RoboDK station: AQIS.rdk

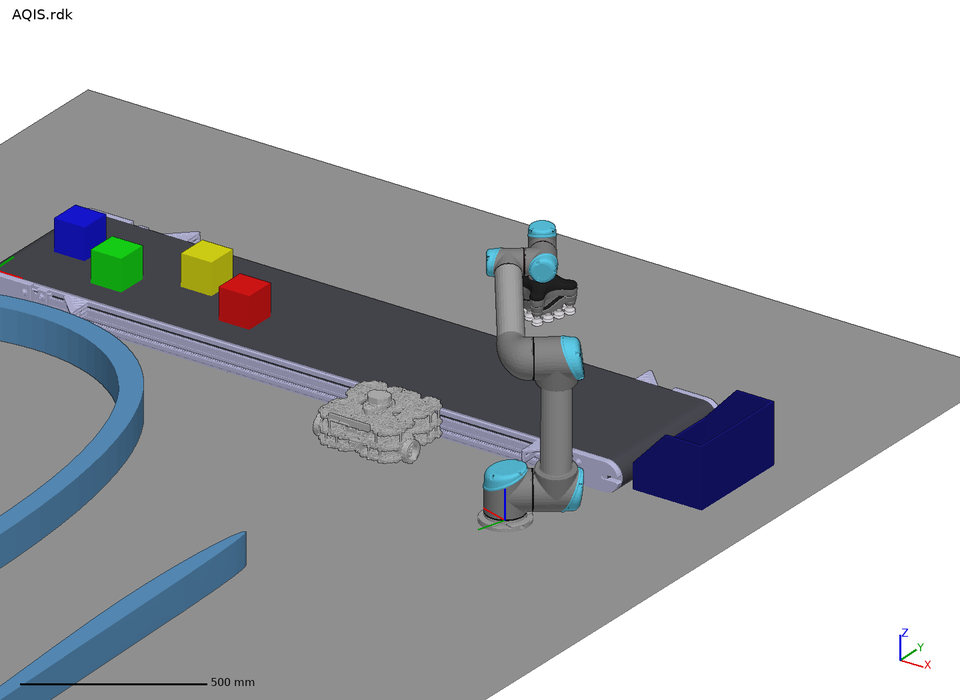
[picture v0: the station drawn from its stored meshes, robots at their saved joint values, targets as dots, program paths as lines]
Station AQIS (saved by RoboDK 5.7.4). Poses are relative to the parent item; angles as X-Y-Z fixed-axis rotations.
  - frame Main at (0, 0, 0) mm
    - frame Conveyor Belt (2m) Base at (0, 1000, 20) mm
      - robot Conveyor Belt (2m): 1 axes
          modified DH rows (alpha deg, a mm, theta deg, d mm): 0, 0, 0, 0 linear
          base shift (0, 0, 0) mm, rotated rx 0 ry 90 rz 0 deg
          joint limits [-500000] to [500000]; home [0]; saved at [0]
    - object Bin Blue at (2060, 1370, -70) mm, rotated rx 0 ry 0 rz -180 deg, size 225 x 337.5 x 191.2 mm, geometry from Bin-Blue.sld
    - object Bin Red at (130, -1910, 0) mm, rotated rx 0 ry 0 rz 90 deg, size 225 x 337.5 x 191.2 mm, geometry from Bin-Red.sld
    - object Blue at (120, 1230, 20) mm, size 100 x 100 x 100 mm, geometry from Blue.step
    - object Green at (310, 1130, 20) mm, size 100 x 100 x 100 mm, geometry from Green.step
    - object Red at (720, 1140, 20) mm, size 100 x 100 x 100 mm, geometry from Red.step
    - object Yellow at (520, 1250, 20) mm, size 100 x 100 x 100 mm, geometry from Yellow.step
    - frame UR5 Base at (1880.84, 695.53, -76.85) mm, rotated rx 0 ry 0 rz 163.4 deg
      - robot UR5: 6 axes
          modified DH rows (alpha deg, a mm, theta deg, d mm): 0, 0, 0, 89.2; 90, 0, 180, 0; 0, 425, 0, 0; 0, 392, 0, 109.3; -90, 0, 0, 94.75; 90, 0, 180, 82.5
          joint limits [-360, -360, -360, -360, -360, -360] to [360, 360, 360, 360, 360, 360]; home [0, -90, -90, 0, 90, 0]; saved at [-36.82, -81.705, -83.159, -101.079, 89.606, 237.429]
        - tool OnRobot VG10 Vacuum Gripper, TCP at (0, 0, 120.9) mm, size 145.4 x 145.4 x 118.3 mm
    - object Floor at (960, 710, -80) mm, size 3000 x 3000 x 0 mm, geometry from Floor.sld
    - object turtlebot3_waffle at (1400, 800, 0) mm, rotated rx 0 ry 0 rz -90 deg, size 280.7 x 305.1 x 138.1 mm, geometry from turtlebot3_waffle.step
    - object Floor at (960, -2290, -80) mm, size 3000 x 3000 x 0 mm, geometry from Floor.sld
    - object path at (430, 2260, 0) mm, rotated rx 0 ry 0 rz 90 deg, size 3159.6 x 1446.5 x 100 mm, geometry from path.step
    - object path at (810, -4600, 0) mm, rotated rx 0 ry 0 rz -90 deg, size 3159.6 x 1446.5 x 100 mm, geometry from path.step
